{attribute 'qualified_only'}
{attribute 'strict'}
TYPE E_DetectionMode :
(
    eRising := 0,
    eFalling := 1
);
END_TYPE

(* stored: Version 1.1.0.1
   DUT E_DetectionMode: Id {1d345440-0ee2-071e-0a54-9bfb112a5c40} *)
